TYPE WrappedComponentExample_Status EXTENDS TcoCore.TcoStruct:
STRUCT

		ProgressThrow:INT;
		ActionDescription:STRING;
END_STRUCT
END_TYPE

(* stored: Version 1.1.0.1
   DUT WrappedComponentExample_Status: Id {1446169e-8254-4b04-a25b-29bf15d85784} *)
